FUNCTION_BLOCK ReadUidTask EXTENDS TcoCore.TcoTask
VAR_IN_OUT
    rfidInOut : RfidInOut;
END_VAR
VAR_INPUT
    ActionDesc : STRING(25);
END_VAR

VAR
    _stringBuilder : TcoCore.StringBuilder;
    _state         : INT;
    _coding        : ARRAY[0..7] OF BYTE;
    _index         : INT;
    _hex           : Tc2_System.T_MaxString := '16# ';
    _uidDataLength : UINT                   := 8;

    _eErrorID   : RFID_FB_U.ERROR;
    _noTagFound : BOOL;
    _uid        : Tc2_System.T_MaxString;
END_VAR

IF (THIS^.Execute()) THEN
    THIS^.ThrowWhen(rfidInOut.xError);

    CASE _state OF

        10:
            // Tag vorhanden
            IF NOT rfidInOut.xTP THEN
                THIS^.Messenger.Error
                (
                    _stringBuilder.Append(ActionDesc)
                        .Append('Tag nicht vorhanden bei Leseversuch')
                        .ToString()
                );

                _noTagFound := TRUE;
                ThrowWhen(TRUE);
            ELSE
                _state := 20;
            END_IF
        20:
            //Command setzen
            rfidInOut.eCommand     := command.INVENTORY;
            rfidInOut.uiDataLenght := _uidDataLength;
            _state                 := 30;
        30:
            // Start der Operation
            rfidInOut.xExecute := TRUE;
            _uid               := '';

            _state := 40;
        40:
            // Warte auf Ende Operation
            rfidInOut.myReadData[_index] :=
                (THIS^.rfidInOut.myReadData[_index]);

            IF rfidInOut.xError THEN
                _uid := '--Error--';
            ELSIF rfidInOut.xDone THEN
                FOR _index := 0 TO UINT_TO_INT(rfidInOut.uiDataLenght - 1) DO

                    _uid := Concat
                    (
                        _uid
                        , BYTE_TO_HEXSTR(in := rfidInOut.myReadData[_index], iPrecision := 2, bLoCase := FALSE)
                    );
                END_FOR

                THIS^.DoneWhen(rfidInOut.xDone);
                THIS^.Messenger.Info('Lesen UID erfolgreich');
                _state := 0;
            END_IF
    END_CASE
END_IF

{attribute 'monitoring' := 'call'}
PROPERTY ErrorId : RFID_FB_U.ERROR
GET
{warning disable C0371}
ErrorId := _eErrorID;
END_GET
END_PROPERTY

METHOD PUBLIC FB_init : BOOL
VAR_INPUT
    bInitRetains : BOOL; // if TRUE, the retain variables are initialized (warm start / cold start)
    bInCopyCode  : BOOL; // if TRUE, the instance afterwards gets moved into the copy code (online change)
    ParentObject : ITcoObject;
END_VAR
// This is not clear to me... I from time to time the consumer code does not see 'FB_init' of 'TcoObject', that's why overridden here with super call...
{warning disable C0316}
SUPER^.FB_init(bInitRetains, bInCopyCode, ParentObject);
END_METHOD

(*~
    <docu>
        <summary>
            Executes when task is aborted.
        </summary>
    </docu>
~*)
METHOD PROTECTED OnAbort
{warning disable C0371}
RfidInOut.eCommand := RFID_FB_U.COMMAND.IDLE;
RfidInOut.xExecute := FALSE;
RfidInOut.xAbort   := FALSE;
END_METHOD

(*~
    <docu>
        <summary>
            Executes when task reaches the ```Done``` state .
        </summary>
    </docu>
~*)
METHOD PROTECTED OnDone
{warning disable C0371}
rfidInOut.xExecute := FALSE;
rfidInOut.eCommand := RFID_FB_U.COMMAND.IDLE;
END_METHOD

(*~
    <docu>
        <summary>
            Executes when task reaches the ```Error``` state.
            <para>
                Do not confuse with <see cref="PlcDocu.TcoCore.TcoTask.WhileError()"/>, that is called cyclically until '''Error''' state is left.
            </para>
        </summary>
    </docu>
~*)
METHOD PROTECTED OnError
{warning disable C0371}

IF _noTagFound THEN
    _eErrorID := RFID_FB_U.ERROR.COMMAND_NO_TAG_FOUND;
ELSE
    _eErrorID := rfidInOut.eErrorID;
END_IF

THIS^.Messenger.Build().Append('Rfid Schreib/Lesekopf Fehler : ').Append(to_string(THIS^._eErrorID)).As().AsError();
END_METHOD

(*~
    <docu>
        <summary>
            Executes ones when the task starts (at the moment of transition from the ```Requested``` state into the ```Busy``` state).
        </summary>
    </docu>
~*)
METHOD PROTECTED OnStart
{warning disable C0371}
rfidInOut.eCommand := RFID_FB_U.COMMAND.IDLE;
rfidInOut.xExecute := FALSE;
rfidInOut.xAbort   := FALSE;
_state             := 10;
END_METHOD

(*~
    <docu>
        <summary>
            Restores this instance to the Ready state. Can be called explicitly or from within one of the restore mechanisms.
            <para>
                See also <see cref="PlcDocu.TcoCore.TcoTask.AutoRestorable()"/>
            </para>
        </summary>
    </docu>
~*)
METHOD Restore : ITcoRestorable
{warning disable C0371}
RfidInOut.eCommand := RFID_FB_U.COMMAND.IDLE;
RfidInOut.xExecute := FALSE;
RfidInOut.xAbort   := FALSE;
_eErrorID          := RFID_FB_U.ERROR.NO_ERROR;
SUPER^.Restore();
END_METHOD

PROPERTY Uid : Tc2_System.T_MaxString
GET
Uid := _uId;
END_GET
END_PROPERTY

END_FUNCTION_BLOCK

(* stored: Version 1.1.0.1, ProductVersion 3.1.4024.12
   POU ReadUidTask: Id {9afc1438-72f3-0359-0d5e-5ae786851400}, SpecialFunc None
   Folder Status: Id {f530cd02-ff3a-0441-19a4-7e82bce8432a}
   Folder TcOpen: Id {d95a24e3-1b2b-07fd-3418-f9e71d5998b1}
   Property ErrorId: Id {1e407204-29be-0058-0e61-c4dedc773dd4}
   Get Get: Id {a51997d0-3568-0e88-01cc-0cc43c0349e3}
   Method FB_init: Id {ae61f780-cede-0a6c-1654-d73b277fd50f}
   Method OnAbort: Id {3da76e41-6814-0867-3efb-26d9bce7ea18}
   Method OnDone: Id {d39af901-1596-0596-186f-e182c5594446}
   Method OnError: Id {a170edc6-80d2-0c3e-1e44-de62810e3d45}
   Method OnStart: Id {430e877e-094e-0b68-257f-a24a7ae8985c}
   Method Restore: Id {46bde516-f86f-02c0-3aa4-3a3ecbadb808}
   Property Uid: Id {41d629f9-13c0-07ac-35de-7ab2da59e1e6}
   Get Get: Id {9881cd9d-1041-0695-2d42-2b90b7c57432} *)
